Fanuc KAREL source: kt00551.KL

-- PROVISIONAL review KL for V940-1; original PC SHA256 51588a4456d4f3a4ab496dec00a49d532c533e5231725ffc8229f2a896f234f9
-- Incomplete behavior may be omitted. Consult companion uncertainty JSON. Do not deploy.
PROGRAM KT00551
%NOLOCKGROUP
-- UNRESOLVED_DECL P1 type=000199
-- UNRESOLVED_DECL P2 type=000199
-- UNRESOLVED_DECL OUT type=000106
BEGIN
  -- V9_ZERO_TABLE_METADATA_HINT layout=0001; no indexed target words; source/name/runtime held
  -- UNRESOLVED_PC offsets 5-44; opcodes 49,7E,49,7E,60,7E,4A
  -- UNRESOLVED_PC offsets 49-53; opcodes 7F
END KT00551
